FUNCTION TryConvert_DWORD_TO_LREAL : BOOL
VAR_INPUT
	in : DWORD;
	out : REFERENCE TO LREAL;
END_VAR

out := DWORD_TO_LREAL(in);
TryConvert_DWORD_TO_LREAL := TRUE;

END_FUNCTION

(* stored: Version 1.1.0.1, ProductVersion 3.1.4024.12
   POU TryConvert_DWORD_TO_LREAL: Id {c35440e8-5342-4d62-bbf8-7ff7d116fbd1}, SpecialFunc None *)
